{attribute 'qualified_only'}
{attribute 'strict'}
TYPE limitCoupling :
(
	None,
	FwSw,
	BwSw,
	Both
);
END_TYPE

(* stored: Version 1.1.0.1, ProductVersion 3.1.4020.12
   DUT limitCoupling: Id {7810a9bc-d383-47ea-8dc8-4d10bb134045} *)
